(*			
	RafalOS
	Rafał Osajda		20.11.2025		TC 4024.66
	Moduł przygotowania danych dla Okna głównego w trybie produkcji
*)
FUNCTION_BLOCK FB_MCHMIPrepareDataForScreen_00_01 EXTENDS FB_MCHMIPrepareDataForScreen IMPLEMENTS ITF_MCHMIPrepareDataForScreen
VAR
END_VAR

(*			
	RafalOS
	Rafał Osajda		19.11.2025		TC 4024.66
	Czyści danych przy zmienia ramki po poprzedniej ramce
*)
METHOD PUBLIC ClearAfterScreen : BOOL
VAR_INPUT
END_VAR
SUPER^.ClearAfterScreen ();
END_METHOD

(*			
	RafalOS
	Rafał Osajda		14.11.2025		TC 4024.66
	Metoda przygotowywania danych dla HMI 
	W niej odbywa się odpytywanie właściego elementu przez łącznik
*)
METHOD PUBLIC PrepareDataForHMI : BOOL
VAR_INPUT
END_VAR
SUPER^.PrepareDataForHMI ();
END_METHOD

(*			
	RafalOS
	Rafał Osajda		19.11.2025		TC 4024.66
	Przygotowanie ramki pood tamke do wyświetlenia - tylko przygotowanie a nie przygotowanie danych do wyświetlenia
*)
METHOD PUBLIC PrepareForScreen : BOOL
VAR_INPUT
END_VAR
SUPER^.PrepareForScreen ();
END_METHOD

END_FUNCTION_BLOCK

(* stored: Version 1.1.0.1
   POU FB_MCHMIPrepareDataForScreen_00_01: Id {a0ca5936-6ba8-006d-10ee-898da7480e87}, SpecialFunc None
   Folder ITF_PDFS: Id {17dd2ebe-9e6b-0bf2-3d90-11a3dbaf0234}
   Method ClearAfterScreen: Id {ffbbed22-fbc0-011c-2b53-cbc9b40d31d2}
   Method PrepareDataForHMI: Id {8db44ae2-3122-084a-00ee-804a2e7492c1}
   Method PrepareForScreen: Id {5f024cf0-dfa2-055b-12d3-48362f8d807d} *)
